FUNCTION_BLOCK KeyValueCollectionDisposedEventHandler EXTENDS KeyValueCollectionEventHandler

METHOD PUBLIC HandleEvent
VAR_INPUT
	Event : I_Event;
END_VAR
VAR
	disposedEvent : I_KeyValueCollectionDisposedEvent;
END_VAR
IF __QUERYINTERFACE(Event, disposedEvent) THEN
	_eventReceived := TRUE;
	fromExpected := disposedEvent.Target = expectedOriginator;
END_IF
END_METHOD

END_FUNCTION_BLOCK

(* stored: Version 1.1.0.1, ProductVersion 3.1.4024.12
   POU KeyValueCollectionDisposedEventHandler: Id {f2505a25-52f4-0909-2ef4-8e8c45a9b6e5}, SpecialFunc None
   Method HandleEvent: Id {d752e4bc-05b3-0afc-0765-50bae27a9d08} *)
